(* PLC project Unnamed, Unknown Unnamed 1 *)
(* stored: creationDateTime 2025-06-13T16:30:15, modificationDateTime 2025-06-13T16:30:15 *)

CONFIGURATION Config0
  RESOURCE Res0 ON PLC
  END_RESOURCE
END_CONFIGURATION
